PROGRAM Zone_Monitoring
VAR
    fbZoneMonitoring: FB_ZoneMonitoring;
END_VAR

//Zone monitoring is following the same structure and logic as FB_ESSMonitoringBase
fbZoneMonitoring(
    iSafetyProvider := Motion_Safety.fbMotionSafety,
    aErrorID =>,
    aErrorMsg =>,
    nAlarmGrpBitNumber =>);

END_PROGRAM

(* stored: Version 1.1.0.1
   POU Zone_Monitoring: Id {f5c11ad1-e7e7-0681-38ec-64bec41cdfdc}, SpecialFunc None *)
